ABB RAPID module: Wobj_FRAME_BufferA.mod

MODULE Wobj_FRAME_BufferA
	! Points are read in order of declaration.
  ! Please do not change the order of points!

  LOCAL PERS robtarget pWobj_U_PointX1:=[[-1265.157,1438.464,160.8819],[0.0527531020343304,-0.892506003379822,0.447874277830124,0.00766136962920427],[1,-1,0,0],[9E+09,9E+09,9E+09,9E+09,9E+09,9E+09]];
	LOCAL PERS robtarget pWobj_U_PointX2:=[[1133.77,1469.633,159.5959],[0.0527557134628296,-0.89251172542572,0.44786274433136,0.00765837728977203],[0,0,-1,0],[9E+09,9E+09,9E+09,9E+09,9E+09,9E+09]];
	LOCAL PERS robtarget pWobj_U_PointY1:=[[-1272.059,2636.979,161.3223],[0.0527618043124676,-0.892510116100311,0.44786536693573,0.00764623889699578],[1,-1,-1,0],[9E+09,9E+09,9E+09,9E+09,9E+09,9E+09]];

ENDMODULE
